// TIA Portal V17 export
// export: Created 2026-04-13T11:12:41.2375706Z, ExportSetting WithDefaults, DisplayName Totally Integrated Automation Portal, DisplayVersion V17 Update 4, DisplayName TIA Portal Openness, DisplayVersion V17 Update 4, DisplayName TIA Portal Version Control Interface, DisplayVersion V17, DisplayName SINAMICS Startdrive Advanced, DisplayVersion V17, DisplayName SINAMICS Startdrive G130, G150, S120, S150, SINAMICS MV, S210, DisplayVersion V17, DisplayName SINAMICS Startdrive G110M, G120, G120C, G120D, G120P, G115D, DisplayVersion V17, DisplayName STEP 7 Professional, DisplayVersion V17 Update 4, DisplayName STEP 7 Safety, DisplayVersion V17, DisplayName WinCC Professional, DisplayVersion V17 Update 4
DATA_BLOCK "INCIP"   // DB10
{ S7_Optimized_Access := 'TRUE' }
VERSION : 0.1
// stored: AutoNumber true, DBAccessibleFromOPCUA true, DBAccessibleFromWebserver true, IsOnlyStoredInLoadMemory false, IsRetainMemResEnabled false, IsWriteProtectedInAS false, MemoryReserve 100
   VAR
      DD电导合格值 : Real;
      JX碱洗温度设定 : Real := 80.0;
      DD电导率当前值 : Real;
      JX碱洗温度 : Real;
      CIP压力 : Real;
      MZD自动清洗 : Bool;
      MSD手动_纯水清洗 : Bool;
      MSD手动_碱水清洗 : Bool;
      MSD手动_溶剂清洗 : Bool;
      MSD手动_热水清洗 : Bool;
      MQX清洗重置 : Bool;
      MCS纯水罐阀门 : Bool;
      MJS碱水罐阀门 : Bool;
      MZS注射水阀门 : Bool;
      MYK压空吹干阀 : Bool;
      MD清洗失败 : Bool;
      MQX室内清洗辅助 : Bool;
      MZT主塔清洗头 : Bool;
      MZT中途停止 : Bool;
      MXT心跳信号发送 : Bool;
      MXT心跳信号接受 : Bool;
      MXY泄压请求 : Bool;
      MGS供水泵请求 : Bool;
      MCIP远程状态 : Bool;
      QCS纯水罐阀门 : Bool;
      QJS碱水罐阀门 : Bool;
      QZS注射水罐阀门 : Bool;
      QYG压干阀门 : Bool;
      QGS供水泵状态CIP : Bool;
      QXY泄压阀门 : Bool;
      PS排水时间 : Real;
      PS排水时间计时 : Real;
   END_VAR
BEGIN
END_DATA_BLOCK
